% RSLogix 500 project Project_11.RSS, saved by version 8.30.00.16 %
PROJECT "UNTITLED"    % processor: Bul.1763 MicroLogix 1100 Series B %

PROGRAM FILES
  LAD 2 "MAIN"  6 rungs
  LAD 3 "IO"  14 rungs  %  I/O -- Read Inputs %
  LAD 4 "DUTY_ROT"  9 rungs  %  Duty Rotation & Assist Staging %
  LAD 5 "ALARMS"  18 rungs  % Alarms %
  LAD 6 "RUN_COMNDS"  3 rungs  % Run Commands %

DATA FILES
  O0 OUTPUT  4 elements
  I1 INPUT  6 elements
  S2 STATUS  66 elements
  B3 BINARY  20 elements
  T4 TIMER  5 elements
  C5 COUNTER  1 elements
  R6 CONTROL  1 elements
  N7 INTEGER  1 elements
  F8 FLOAT  1 elements

LADDER 2 "MAIN"
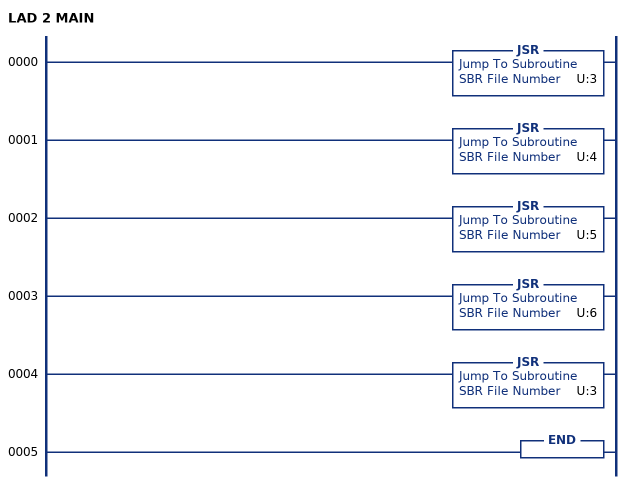
% Rung: 0 %
SOR JSR U:3 EOR
% Rung: 1 %
SOR JSR U:4 EOR
% Rung: 2 %
SOR JSR U:5 EOR
% Rung: 3 %
SOR JSR U:6 EOR
% Rung: 4 %
SOR JSR U:3 EOR
% Rung: 5 %
SOR END EOR

LADDER 3 "IO"    %  I/O -- Read Inputs %
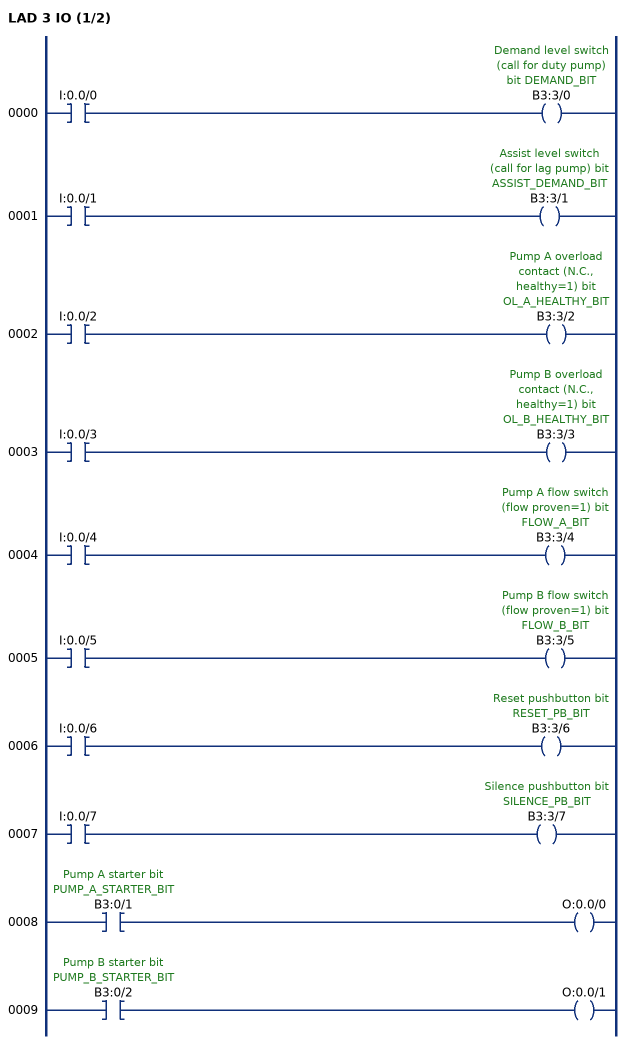
% Rung: 0 %
SOR XIC I:0.0/0 OTE B3:3/0 EOR
%   B3:3/0  DEMAND_BIT  "Demand level switch (call for duty pump) bit" %
% Rung: 1 %
SOR XIC I:0.0/1 OTE B3:3/1 EOR
%   B3:3/1  ASSIST_DEMAND_BIT  "Assist level switch (call for lag pump) bit" %
% Rung: 2 %
SOR XIC I:0.0/2 OTE B3:3/2 EOR
%   B3:3/2  OL_A_HEALTHY_BIT  "Pump A overload contact (N.C., healthy=1) bit" %
% Rung: 3 %
SOR XIC I:0.0/3 OTE B3:3/3 EOR
%   B3:3/3  OL_B_HEALTHY_BIT  "Pump B overload contact (N.C., healthy=1) bit" %
% Rung: 4 %
SOR XIC I:0.0/4 OTE B3:3/4 EOR
%   B3:3/4  FLOW_A_BIT  "Pump A flow switch (flow proven=1) bit" %
% Rung: 5 %
SOR XIC I:0.0/5 OTE B3:3/5 EOR
%   B3:3/5  FLOW_B_BIT  "Pump B flow switch (flow proven=1) bit" %
% Rung: 6 %
SOR XIC I:0.0/6 OTE B3:3/6 EOR
%   B3:3/6  RESET_PB_BIT  "Reset pushbutton bit" %
% Rung: 7 %
SOR XIC I:0.0/7 OTE B3:3/7 EOR
%   B3:3/7  SILENCE_PB_BIT  "Silence pushbutton bit" %
% Rung: 8 %
SOR XIC B3:0/1 OTE O:0.0/0 EOR
%   B3:0/1  PUMP_A_STARTER_BIT  "Pump A starter bit" %
% Rung: 9 %
SOR XIC B3:0/2 OTE O:0.0/1 EOR
%   B3:0/2  PUMP_B_STARTER_BIT  "Pump B starter bit" %

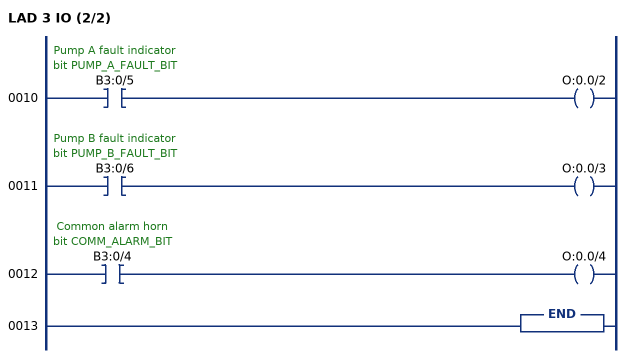
% Rung: 10 %
SOR XIC B3:0/5 OTE O:0.0/2 EOR
%   B3:0/5  PUMP_A_FAULT_BIT  "Pump A fault indicator bit" %
% Rung: 11 %
SOR XIC B3:0/6 OTE O:0.0/3 EOR
%   B3:0/6  PUMP_B_FAULT_BIT  "Pump B fault indicator bit" %
% Rung: 12 %
SOR XIC B3:0/4 OTE O:0.0/4 EOR
%   B3:0/4  COMM_ALARM_BIT  "Common alarm horn bit" %
% Rung: 13 %
SOR END EOR

LADDER 4 "DUTY_ROT"    %  Duty Rotation & Assist Staging %
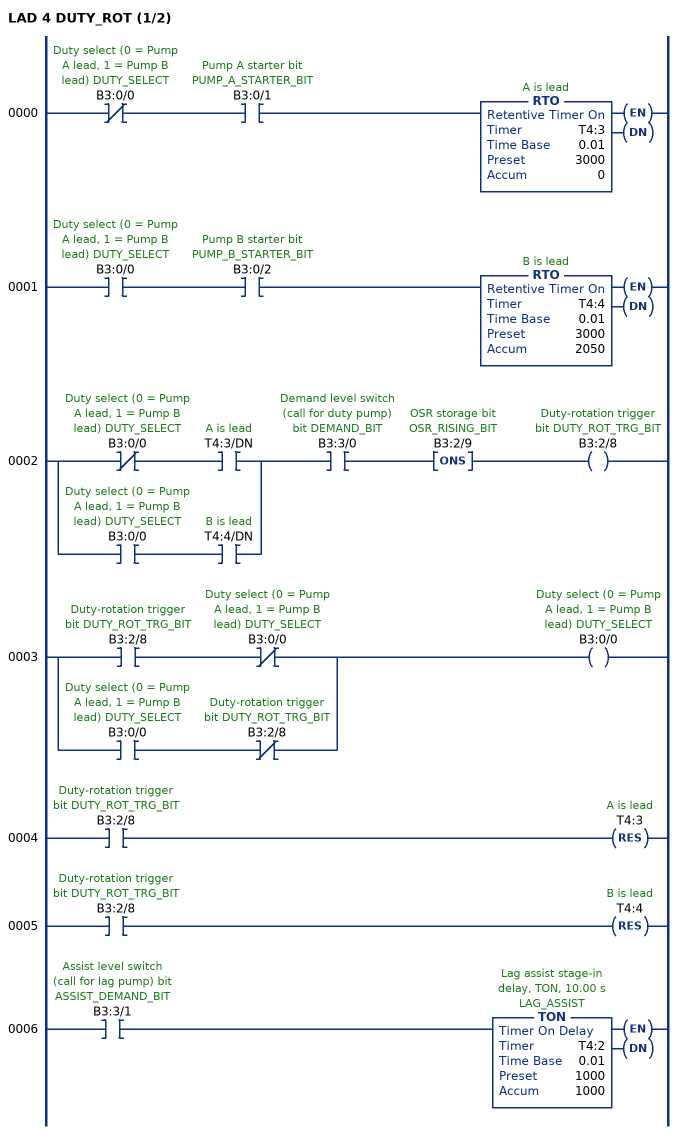
% Rung: 0 %
SOR XIO B3:0/0 XIC B3:0/1 RTO T4:3 0.01 3000 0 EOR
%   B3:0/0  DUTY_SELECT  "Duty select (0 = Pump A lead, 1 = Pump B lead)" %
%   B3:0/1  PUMP_A_STARTER_BIT  "Pump A starter bit" %
%   T4:3  "A is lead" %
% Rung: 1 %
SOR XIC B3:0/0 XIC B3:0/2 RTO T4:4 0.01 3000 2050 EOR
%   B3:0/0  DUTY_SELECT  "Duty select (0 = Pump A lead, 1 = Pump B lead)" %
%   B3:0/2  PUMP_B_STARTER_BIT  "Pump B starter bit" %
%   T4:4  "B is lead" %
% Rung: 2 %
SOR BST XIO B3:0/0 XIC T4:3/DN NXB XIC B3:0/0 XIC T4:4/DN BND XIC B3:3/0 ONS B3:2/9 OTE B3:2/8 EOR
%   B3:0/0  DUTY_SELECT  "Duty select (0 = Pump A lead, 1 = Pump B lead)" %
%   T4:3  "A is lead" %
%   T4:4  "B is lead" %
%   B3:3/0  DEMAND_BIT  "Demand level switch (call for duty pump) bit" %
%   B3:2/9  OSR_RISING_BIT  "OSR storage bit" %
%   B3:2/8  DUTY_ROT_TRG_BIT  "Duty-rotation trigger bit" %
% Rung: 3 %
SOR BST XIC B3:2/8 XIO B3:0/0 NXB XIC B3:0/0 XIO B3:2/8 BND OTE B3:0/0 EOR
%   B3:2/8  DUTY_ROT_TRG_BIT  "Duty-rotation trigger bit" %
%   B3:0/0  DUTY_SELECT  "Duty select (0 = Pump A lead, 1 = Pump B lead)" %
% Rung: 4 %
SOR XIC B3:2/8 RES T4:3 EOR
%   B3:2/8  DUTY_ROT_TRG_BIT  "Duty-rotation trigger bit" %
%   T4:3  "A is lead" %
% Rung: 5 %
SOR XIC B3:2/8 RES T4:4 EOR
%   B3:2/8  DUTY_ROT_TRG_BIT  "Duty-rotation trigger bit" %
%   T4:4  "B is lead" %
% Rung: 6 %
SOR XIC B3:3/1 TON T4:2 0.01 1000 1000 EOR
%   B3:3/1  ASSIST_DEMAND_BIT  "Assist level switch (call for lag pump) bit" %
%   T4:2  LAG_ASSIST  "Lag assist stage-in delay, TON, 10.00 s" %

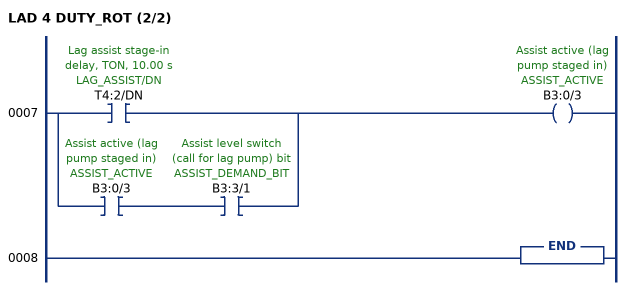
% Rung: 7 %
SOR BST XIC T4:2/DN NXB XIC B3:0/3 XIC B3:3/1 BND OTE B3:0/3 EOR
%   T4:2  LAG_ASSIST  "Lag assist stage-in delay, TON, 10.00 s" %
%   B3:0/3  ASSIST_ACTIVE  "Assist active (lag pump staged in)" %
%   B3:3/1  ASSIST_DEMAND_BIT  "Assist level switch (call for lag pump) bit" %
% Rung: 8 %
SOR END EOR

LADDER 5 "ALARMS"    % Alarms %
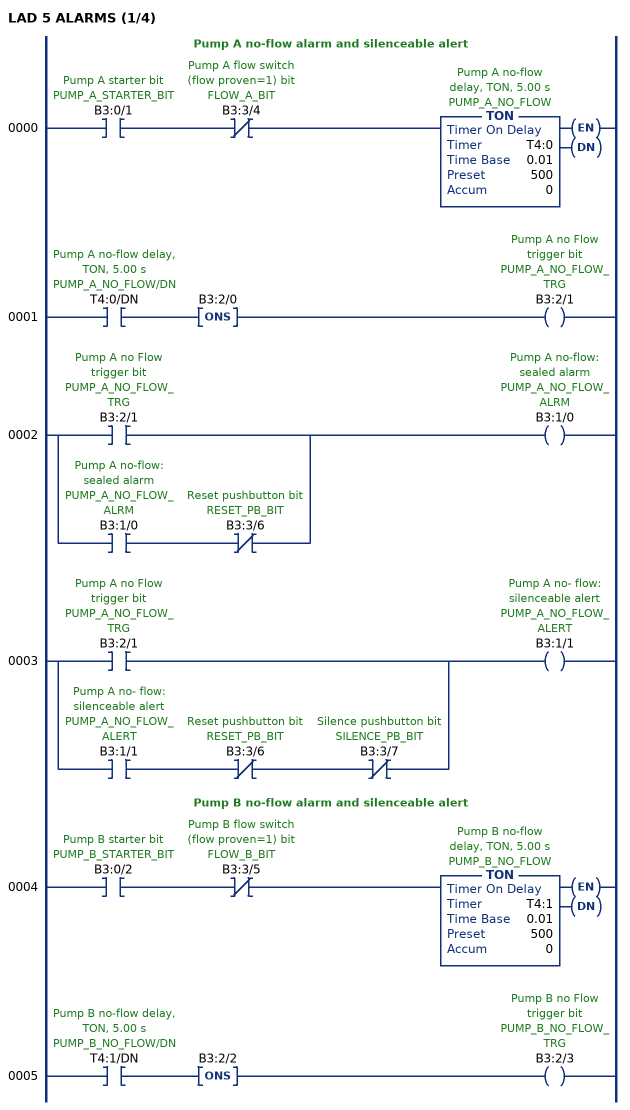
% Rung: 0 %
% TITLE: Pump A no-flow alarm and silenceable alert %
SOR XIC B3:0/1 XIO B3:3/4 TON T4:0 0.01 500 0 EOR
%   B3:0/1  PUMP_A_STARTER_BIT  "Pump A starter bit" %
%   B3:3/4  FLOW_A_BIT  "Pump A flow switch (flow proven=1) bit" %
%   T4:0  PUMP_A_NO_FLOW  "Pump A no-flow delay, TON, 5.00 s" %
% Rung: 1 %
SOR XIC T4:0/DN ONS B3:2/0 OTE B3:2/1 EOR
%   T4:0  PUMP_A_NO_FLOW  "Pump A no-flow delay, TON, 5.00 s" %
%   B3:2/1  PUMP_A_NO_FLOW_TRG  "Pump A no Flow trigger bit" %
% Rung: 2 %
SOR BST XIC B3:2/1 NXB XIC B3:1/0 XIO B3:3/6 BND OTE B3:1/0 EOR
%   B3:2/1  PUMP_A_NO_FLOW_TRG  "Pump A no Flow trigger bit" %
%   B3:1/0  PUMP_A_NO_FLOW_ALRM  "Pump A no-flow: sealed alarm" %
%   B3:3/6  RESET_PB_BIT  "Reset pushbutton bit" %
% Rung: 3 %
SOR BST XIC B3:2/1 NXB XIC B3:1/1 XIO B3:3/6 XIO B3:3/7 BND OTE B3:1/1 EOR
%   B3:2/1  PUMP_A_NO_FLOW_TRG  "Pump A no Flow trigger bit" %
%   B3:1/1  PUMP_A_NO_FLOW_ALERT  "Pump A no- flow: silenceable alert" %
%   B3:3/6  RESET_PB_BIT  "Reset pushbutton bit" %
%   B3:3/7  SILENCE_PB_BIT  "Silence pushbutton bit" %
% Rung: 4 %
% TITLE: Pump B no-flow alarm and silenceable alert %
SOR XIC B3:0/2 XIO B3:3/5 TON T4:1 0.01 500 0 EOR
%   B3:0/2  PUMP_B_STARTER_BIT  "Pump B starter bit" %
%   B3:3/5  FLOW_B_BIT  "Pump B flow switch (flow proven=1) bit" %
%   T4:1  PUMP_B_NO_FLOW  "Pump B no-flow delay, TON, 5.00 s" %
% Rung: 5 %
SOR XIC T4:1/DN ONS B3:2/2 OTE B3:2/3 EOR
%   T4:1  PUMP_B_NO_FLOW  "Pump B no-flow delay, TON, 5.00 s" %
%   B3:2/3  PUMP_B_NO_FLOW_TRG  "Pump B no Flow trigger bit" %

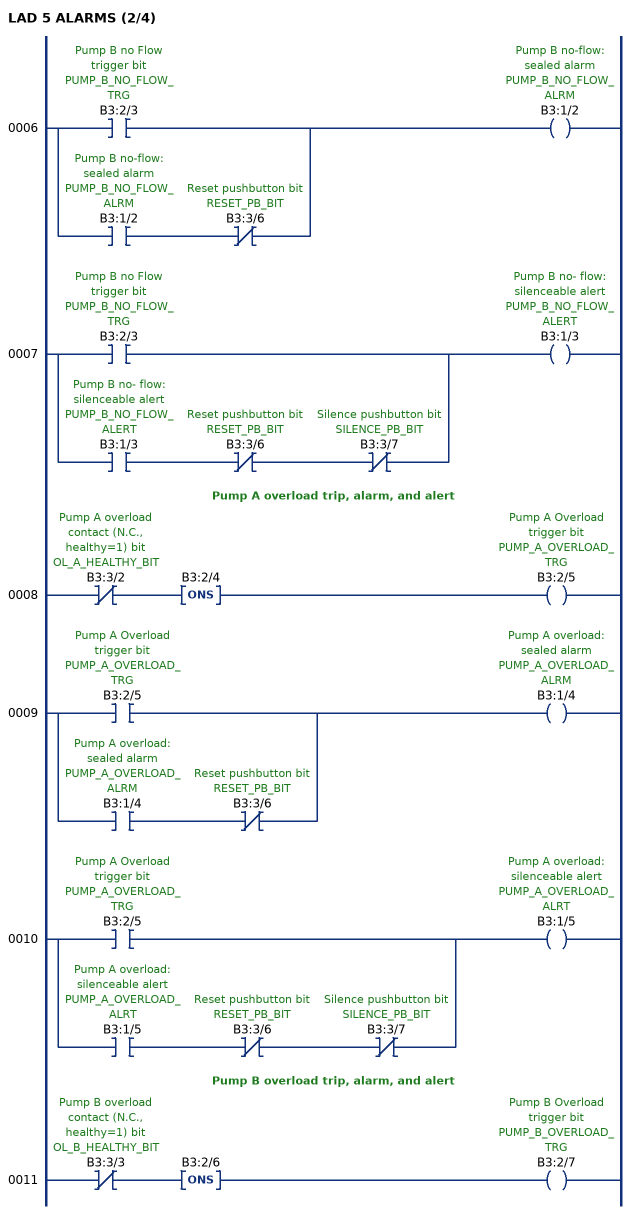
% Rung: 6 %
SOR BST XIC B3:2/3 NXB XIC B3:1/2 XIO B3:3/6 BND OTE B3:1/2 EOR
%   B3:2/3  PUMP_B_NO_FLOW_TRG  "Pump B no Flow trigger bit" %
%   B3:1/2  PUMP_B_NO_FLOW_ALRM  "Pump B no-flow: sealed alarm" %
%   B3:3/6  RESET_PB_BIT  "Reset pushbutton bit" %
% Rung: 7 %
SOR BST XIC B3:2/3 NXB XIC B3:1/3 XIO B3:3/6 XIO B3:3/7 BND OTE B3:1/3 EOR
%   B3:2/3  PUMP_B_NO_FLOW_TRG  "Pump B no Flow trigger bit" %
%   B3:1/3  PUMP_B_NO_FLOW_ALERT  "Pump B no- flow: silenceable alert" %
%   B3:3/6  RESET_PB_BIT  "Reset pushbutton bit" %
%   B3:3/7  SILENCE_PB_BIT  "Silence pushbutton bit" %
% Rung: 8 %
% TITLE: Pump A overload trip, alarm, and alert %
SOR XIO B3:3/2 ONS B3:2/4 OTE B3:2/5 EOR
%   B3:3/2  OL_A_HEALTHY_BIT  "Pump A overload contact (N.C., healthy=1) bit" %
%   B3:2/5  PUMP_A_OVERLOAD_TRG  "Pump A Overload trigger bit" %
% Rung: 9 %
SOR BST XIC B3:2/5 NXB XIC B3:1/4 XIO B3:3/6 BND OTE B3:1/4 EOR
%   B3:2/5  PUMP_A_OVERLOAD_TRG  "Pump A Overload trigger bit" %
%   B3:1/4  PUMP_A_OVERLOAD_ALRM  "Pump A overload: sealed alarm" %
%   B3:3/6  RESET_PB_BIT  "Reset pushbutton bit" %
% Rung: 10 %
SOR BST XIC B3:2/5 NXB XIC B3:1/5 XIO B3:3/6 XIO B3:3/7 BND OTE B3:1/5 EOR
%   B3:2/5  PUMP_A_OVERLOAD_TRG  "Pump A Overload trigger bit" %
%   B3:1/5  PUMP_A_OVERLOAD_ALRT  "Pump A overload: silenceable alert" %
%   B3:3/6  RESET_PB_BIT  "Reset pushbutton bit" %
%   B3:3/7  SILENCE_PB_BIT  "Silence pushbutton bit" %
% Rung: 11 %
% TITLE: Pump B overload trip, alarm, and alert %
SOR XIO B3:3/3 ONS B3:2/6 OTE B3:2/7 EOR
%   B3:3/3  OL_B_HEALTHY_BIT  "Pump B overload contact (N.C., healthy=1) bit" %
%   B3:2/7  PUMP_B_OVERLOAD_TRG  "Pump B Overload trigger bit" %

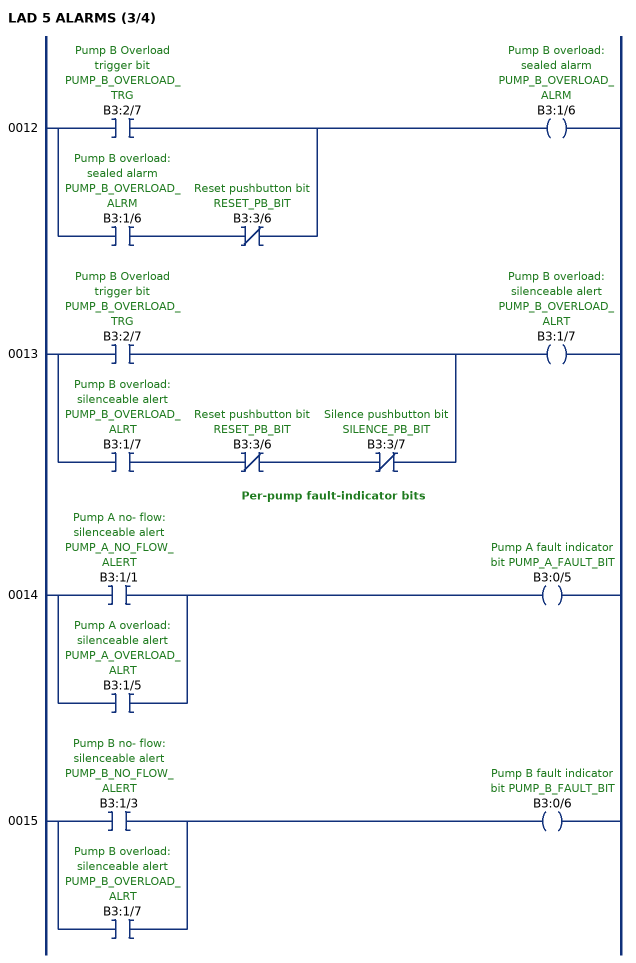
% Rung: 12 %
SOR BST XIC B3:2/7 NXB XIC B3:1/6 XIO B3:3/6 BND OTE B3:1/6 EOR
%   B3:2/7  PUMP_B_OVERLOAD_TRG  "Pump B Overload trigger bit" %
%   B3:1/6  PUMP_B_OVERLOAD_ALRM  "Pump B overload: sealed alarm" %
%   B3:3/6  RESET_PB_BIT  "Reset pushbutton bit" %
% Rung: 13 %
SOR BST XIC B3:2/7 NXB XIC B3:1/7 XIO B3:3/6 XIO B3:3/7 BND OTE B3:1/7 EOR
%   B3:2/7  PUMP_B_OVERLOAD_TRG  "Pump B Overload trigger bit" %
%   B3:1/7  PUMP_B_OVERLOAD_ALRT  "Pump B overload: silenceable alert" %
%   B3:3/6  RESET_PB_BIT  "Reset pushbutton bit" %
%   B3:3/7  SILENCE_PB_BIT  "Silence pushbutton bit" %
% Rung: 14 %
% TITLE: Per-pump fault-indicator bits %
SOR BST XIC B3:1/1 NXB XIC B3:1/5 BND OTE B3:0/5 EOR
%   B3:1/1  PUMP_A_NO_FLOW_ALERT  "Pump A no- flow: silenceable alert" %
%   B3:1/5  PUMP_A_OVERLOAD_ALRT  "Pump A overload: silenceable alert" %
%   B3:0/5  PUMP_A_FAULT_BIT  "Pump A fault indicator bit" %
% Rung: 15 %
SOR BST XIC B3:1/3 NXB XIC B3:1/7 BND OTE B3:0/6 EOR
%   B3:1/3  PUMP_B_NO_FLOW_ALERT  "Pump B no- flow: silenceable alert" %
%   B3:1/7  PUMP_B_OVERLOAD_ALRT  "Pump B overload: silenceable alert" %
%   B3:0/6  PUMP_B_FAULT_BIT  "Pump B fault indicator bit" %

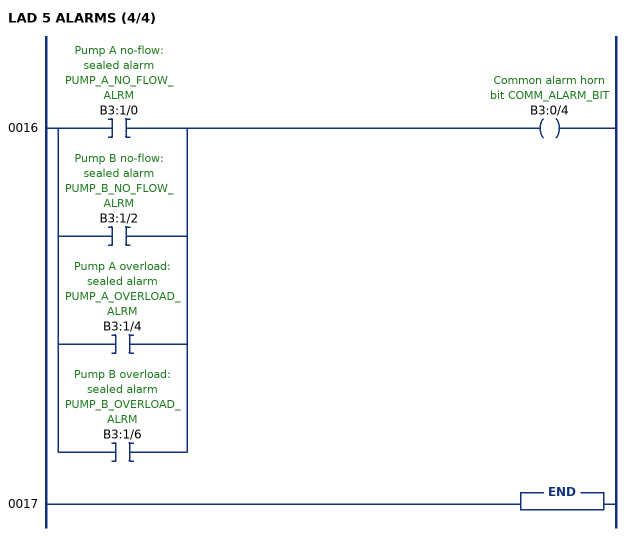
% Rung: 16 %
SOR BST XIC B3:1/0 NXB XIC B3:1/2 NXB XIC B3:1/4 NXB XIC B3:1/6 BND OTE B3:0/4 EOR
%   B3:1/0  PUMP_A_NO_FLOW_ALRM  "Pump A no-flow: sealed alarm" %
%   B3:1/2  PUMP_B_NO_FLOW_ALRM  "Pump B no-flow: sealed alarm" %
%   B3:1/4  PUMP_A_OVERLOAD_ALRM  "Pump A overload: sealed alarm" %
%   B3:1/6  PUMP_B_OVERLOAD_ALRM  "Pump B overload: sealed alarm" %
%   B3:0/4  COMM_ALARM_BIT  "Common alarm horn bit" %
% Rung: 17 %
SOR END EOR

LADDER 6 "RUN_COMNDS"    % Run Commands %
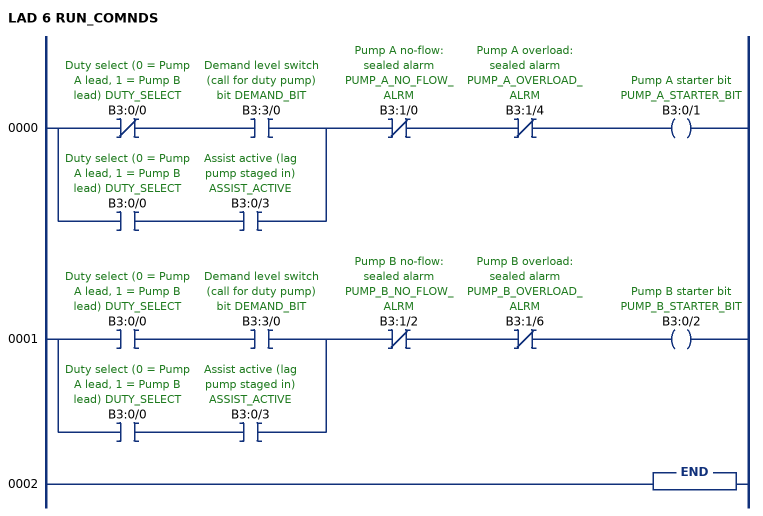
% Rung: 0 %
SOR BST XIO B3:0/0 XIC B3:3/0 NXB XIC B3:0/0 XIC B3:0/3 BND XIO B3:1/0 XIO B3:1/4 OTE B3:0/1 EOR
%   B3:0/0  DUTY_SELECT  "Duty select (0 = Pump A lead, 1 = Pump B lead)" %
%   B3:3/0  DEMAND_BIT  "Demand level switch (call for duty pump) bit" %
%   B3:0/3  ASSIST_ACTIVE  "Assist active (lag pump staged in)" %
%   B3:1/0  PUMP_A_NO_FLOW_ALRM  "Pump A no-flow: sealed alarm" %
%   B3:1/4  PUMP_A_OVERLOAD_ALRM  "Pump A overload: sealed alarm" %
%   B3:0/1  PUMP_A_STARTER_BIT  "Pump A starter bit" %
% Rung: 1 %
SOR BST XIC B3:0/0 XIC B3:3/0 NXB XIC B3:0/0 XIC B3:0/3 BND XIO B3:1/2 XIO B3:1/6 OTE B3:0/2 EOR
%   B3:0/0  DUTY_SELECT  "Duty select (0 = Pump A lead, 1 = Pump B lead)" %
%   B3:3/0  DEMAND_BIT  "Demand level switch (call for duty pump) bit" %
%   B3:0/3  ASSIST_ACTIVE  "Assist active (lag pump staged in)" %
%   B3:1/2  PUMP_B_NO_FLOW_ALRM  "Pump B no-flow: sealed alarm" %
%   B3:1/6  PUMP_B_OVERLOAD_ALRM  "Pump B overload: sealed alarm" %
%   B3:0/2  PUMP_B_STARTER_BIT  "Pump B starter bit" %
% Rung: 2 %
SOR END EOR

OTHER DOCUMENTED ADDRESSES
  PFILE:7  "I/O -- Write Output s"

DATA TABLE (non-zero values as saved)
DATA B3
% B3:0 % 0X000F 0X0000 0X0000 0X003F 0X0000 0X0000 0X0000 0X0000 0X0000 0X0000
DATA T4
% .PRE .ACC %
% T4:0 % 500 0
% T4:1 % 500 0
% T4:2 % 1000 1000
% T4:3 % 3000 0
% T4:4 % 3000 2050
